// TwinCAT 3 PLC project Solutions
// ProgramVersion: 3.1.4026.11
// libraries:
//   CNM_AbstractObject, * (ekvip automation GmbH)
//   CNM AoC Lib, * (ekvip automation GmbH)
//   CNM_AssertionInterfaceLib, * (ekvip automation GmbH)
//   CNM_CollectionInterfaces, * (ekvip automation GmbH)
//   CNM_Collections, * (ekvip automation GmbH)
//   CNM_CycleManager, * (ekvip automation GmbH)
//   CNM_CylceManagerInterfaces, * (ekvip automation GmbH)
//   CNM_ReturnTypes, * (ekvip automation GmbH)
//   CNM_UnicodeUtilities, * (ekvip automation GmbH)
//   Tc2_Standard, * (Beckhoff Automation GmbH)
//   Tc2_System, * (Beckhoff Automation GmbH)
// project tree:
//   Day01/ Day01Solution.TcPOU
//   Day02/ Day02Solution.TcPOU
//   Day06/Guard/ Guard.TcPOU, IGuard.TcIO
//   Day06/Moves/ GuardMove.TcPOU, IMove.TcIO, MoveUp.TcPOU, MoveRight.TcPOU, MoveDown.TcPOU, MoveLeft.TcPOU
//   Day06/ Rotation.TcDUT, Day06Solution.TcPOU
//   Day07/ Day07Solution.TcPOU
//   Day05/ Day05Solution.TcPOU, IPage.TcIO, Page.TcPOU
//   Day04/ CharObj.TcPOU, Day04Solution.TcPOU, IChar.TcIO
//   Day03/ Day03Solution.TcPOU, DontInstruction.TcPOU, ISumCollectorLINT.TcIO, MulInstruction.TcPOU, DoInstruction.TcPOU, SumCollectorLINT.TcPOU
//   Helpers/DynArray/ Dynamic2dArray.TcPOU, I2dArray.TcIO
//   Parsers/ NumberParser.TcPOU
//   / PlcTask.TcTTO
//   POUs/ LocalIoAddresses.TcGVL, MAIN.TcPOU
// real-time tasks:
//   TASK PlcTask: cycle T#10ms, priority 20, ADS port 350

CONFIGURATION Solutions
    RESOURCE PLC ON TwinCAT3
        TASK PlcTask(INTERVAL := T#10ms, PRIORITY := 20);
        PROGRAM MAIN WITH PlcTask : MAIN;
    END_RESOURCE
END_CONFIGURATION

// ---- Day06/Rotation.TcDUT
{attribute 'qualified_only'}
{attribute 'strict'}
TYPE Rotation :
(
	UP := 0,
	RIGHT := 1,
	DOWN := 2,
	LEFT := 3
)DINT;
END_TYPE

// ---- POUs/LocalIoAddresses.TcGVL
{attribute 'qualified_only'}
VAR_GLOBAL
	NetId :STRING := '10.175.16.49.1.1';
	Path :STRING := 'C:\Users\tdie\Documents\tdie_AOC\2024';
END_VAR

// ---- Day06/Guard/IGuard.TcIO
INTERFACE IGuard

PROPERTY direction : Rotation
GET
END_GET
SET
END_SET
END_PROPERTY

METHOD walk
VAR_INPUT
	map :I2dArray;
END_VAR
END_METHOD

PROPERTY x : DINT
GET
END_GET
SET
END_SET
END_PROPERTY

PROPERTY y : DINT
GET
END_GET
SET
END_SET
END_PROPERTY

END_INTERFACE

// ---- Day06/Moves/IMove.TcIO
INTERFACE IMove

METHOD tryMove : BOOL
VAR_INPUT
	guard :IGuard;
	map :I2dArray;
	collision :DINT := 1;
END_VAR
END_METHOD

END_INTERFACE

// ---- Day03/ISumCollectorLINT.TcIO
INTERFACE ISumCollectorLINT EXTENDS CNM_AbstractObject.IObject

METHOD addValue
VAR_INPUT
	value :LINT;
END_VAR
END_METHOD

PROPERTY enabled : BOOL
GET
END_GET
SET
END_SET
END_PROPERTY

PROPERTY sum : LINT
GET
END_GET
SET
END_SET
END_PROPERTY

END_INTERFACE

// ---- Day04/IChar.TcIO
INTERFACE IChar EXTENDS IObject

PROPERTY charAsByte : Byte
GET
END_GET
END_PROPERTY

PROPERTY charAsString : STRING(1)
GET
END_GET
END_PROPERTY

END_INTERFACE

// ---- Day05/IPage.TcIO
INTERFACE IPage EXTENDS IObject, CNM_AoC.IHaveValue

METHOD addSuccessor
VAR_INPUT
	successor :CNM_AoC.IHaveValue;
END_VAR
END_METHOD

END_INTERFACE

// ---- Helpers/DynArray/I2dArray.TcIO
INTERFACE I2dArray EXTENDS CNM_AbstractObject.IObject

METHOD getObjectAt : IObject
VAR_INPUT
	y :UDINT; //dimension 1
	x :UDINT; //dimension 2
END_VAR
END_METHOD

METHOD isInBounds : BOOL
VAR_INPUT
	x :UDINT;
	y :UDINT;
END_VAR
END_METHOD

METHOD setObjectAt
VAR_INPUT
	y :UDINT; //dimension 1
	x :UDINT; //dimension 2
	obj :CNM_AbstractObject.IObject;
END_VAR
END_METHOD

END_INTERFACE

// ---- POUs/MAIN.TcPOU
PROGRAM MAIN
VAR
	day01 :Day01Solution(sNetId := LocalIoAddresses.NetId, folderPath := LocalIoAddresses.Path, inputFile := 'day01.txt', outputFile := 'solution.txt');
	day02 :Day02Solution(sNetId := LocalIoAddresses.NetId, folderPath := LocalIoAddresses.Path, inputFile := 'day02.txt', outputFile := 'solution.txt');
	day03 :Day03Solution(sNetId := LocalIoAddresses.NetId, folderPath := LocalIoAddresses.Path, inputFile := 'day03.txt', outputFile := 'solution.txt');
	day04 :Day04Solution(sNetId := LocalIoAddresses.NetId, folderPath := LocalIoAddresses.Path, inputFile := 'day04.txt', outputFile := 'solution.txt');
	day05 :Day05Solution(sNetId := LocalIoAddresses.NetId, folderPath := LocalIoAddresses.Path, inputFile := 'day05.txt', outputFile := 'solution.txt');
	day06 :Day06Solution(sNetId := LocalIoAddresses.NetId, folderPath := LocalIoAddresses.Path, inputFile := 'day06.txt', outputFile := 'solution.txt');
	day07 :Day07Solution(sNetId := LocalIoAddresses.NetId, folderPath := LocalIoAddresses.Path, inputFile := 'day07.txt', outputFile := 'solution.txt');
END_VAR

//some are really slow because I do to few operations each cycle, might take up to 30 seconds to complete!
day01.run(FALSE);
day02.run(FALSE);
day03.run(FALSE); 
day04.run(FALSE); 
day05.run(FALSE); 
day06.run(FALSE); 
day07.run(FALSE);

END_PROGRAM

// ---- Day01/Day01Solution.TcPOU
FUNCTION_BLOCK Day01Solution EXTENDS CNM_AoC.AbstractSolver

METHOD solve
VAR_INPUT
	step	: DINT;
END_VAR
VAR_INST
	pathInserted :BOOL;
	left :CNM_Collections.ArrayList(100);
	right :CNM_Collections.ArrayList(100);
	parser :NumberParser();
	sum : DINT;
END_VAR
VAR
	parsed :CNM_CollectionInterfaces.IArrayList;
	tmpObj :CNM_AbstractObject.IObject;
	value1 :CNM_AoC.IHaveValue;
	value2 :CNM_AoC.IHaveValue;
	index : DINT;
	currentLine :ILine;
	currentLineObject :IObject;
END_VAR
VAR CONSTANT
	READ_INPUT :DINT := 2;
	GET_LINES :DINT := READ_INPUT + 1;
	PARSE :DINT := GET_LINES + 1;
	SORT_LEFT :DINT := PARSE + 1;
	SORT_RIGHT :DINT := SORT_LEFT + 1;
	SOLVE_PART1 :DINT := SORT_RIGHT + 1;
	RESET_FOR_PART2 :DINT := SOLVE_PART1 + 1;
	SOLVE_PART2 :DINT := RESET_FOR_PART2 + 1;
	APPEND_SOLUTION :DINT := SOLVE_PART2 + 1;
	WRITE_SOLUTION :DINT := APPEND_SOLUTION + 1;
	CLEAN_UP :DINT := WRITE_SOLUTION + 1;
END_VAR
CASE step OF
PARSE:	
	THIS^.lines.iterate(execute := FALSE);
	WHILE(THIS^.lines.iterate(execute := TRUE, line => currentLine) = CNM_ReturnTypes.SingleExecutionState.BUSY)DO
		parsed := parser.getAllNumbers(currentLine);
		left.append(parsed.dequeue());
		right.append(parsed.dequeue());
		parsed.deepDestruct();
	END_WHILE
	cm.proceed();
SORT_LEFT:
	cm.evaluate(SEL(right.size = left.size, CNM_ReturnTypes.SingleExecutionState.ERROR, CNM_ReturnTypes.SingleExecutionState.SUCCESS));
	cm.evaluate(left.instant.sort());
SORT_RIGHT:
	cm.evaluate(right.instant.sort());
SOLVE_PART1:
	FOR index := 0 TO TO_DINT(left.size)-1 DO
		left.getObjectAt(index, object => tmpObj);
		__QUERYINTERFACE(tmpObj, value1);
		right.getObjectAt(index, object => tmpObj);
		__QUERYINTERFACE(tmpObj, value2);
		sum := sum + TO_DINT(ABS(value1.value - value2.value));
	END_FOR
	THIS^.bufferWrite := Concat(TO_STRING(sum), '$n');
	cm.proceed();
RESET_FOR_PART2:
	left.iterate(FALSE);
	sum := 0;
	cm.proceed();
SOLVE_PART2:
	cm.evaluate(left.iterate(TRUE, object => tmpObj));
	IF(__QUERYINTERFACE(tmpObj, value1))THEN
		right.iterate(FALSE);
		WHILE(right.iterate(TRUE, object => tmpObj) = CNM_ReturnTypes.SingleExecutionState.BUSY AND __QUERYINTERFACE(tmpObj, value2))DO
			IF(value1.value = value2.value)THEN
				sum := sum + TO_DINT(value1.value);
			END_IF
			IF(value2.value > value1.value)THEN
				EXIT;
			END_IF
		END_WHILE
	END_IF		
APPEND_SOLUTION:
	THIS^.bufferWrite :=Concat(THIS^.bufferWrite, Concat(TO_STRING(sum), '$n'));
	cm.proceed();
WRITE_SOLUTION:
	THIS^.writeSolution();
CLEAN_UP:
	cm.step.next := CNM_ReturnTypes.DefaultSteps.STEP.SUCCESS;
	lines.deepDestruct();
	left.deepDestruct();
	right.deepDestruct();
	cm.proceed();
END_CASE
END_METHOD

END_FUNCTION_BLOCK

// ---- Parsers/NumberParser.TcPOU
FUNCTION_BLOCK NumberParser
VAR_INPUT
END_VAR
VAR_OUTPUT
END_VAR
VAR
END_VAR

METHOD getAllNumbers : IArrayList
VAR_INPUT
	container :CNM_AoC.IStringContainer;
END_VAR
VAR
	index : DINT;
	currentParseValue :DINT;
	currentLineText : STRING(255);
	found :BOOL;
	result :CNM_CollectionInterfaces.IArrayList;
	pResult :POINTER TO CNM_Collections.ArrayList;
	pValue :POINTER TO CNM_AoC.Value;
	value :CNM_AoC.IHaveValue;
END_VAR
pResult := __NEW(ArrayList(initialSize := 2));
__QUERYINTERFACE(pResult^, result);
currentLineText := container.text;

FOR index := 0 TO LEN(container.text)-1 DO
	IF(currentLineText[index] >= 48 AND currentLineText[index] <= 57)THEN
		currentParseValue := currentParseValue * 10;
		currentParseValue := currentParseValue + currentLineText[index]-48;
		found := TRUE;
	ELSE
		IF(found)THEN
			pValue := __NEW(Value);
			__QUERYINTERFACE(pValue^, value);
			value.value := currentParseValue;//add num to result
			result.append(value);
		END_IF
		currentParseValue := 0;
		found := FALSE;
	END_IF
END_FOR	

IF(found)THEN
	pValue := __NEW(Value);
	__QUERYINTERFACE(pValue^, value);
	value.value := currentParseValue;//add num to result
	result.append(value);
END_IF

getAllNumbers := result;
END_METHOD

METHOD getAllNumbersLint : IArrayList
VAR_INPUT
	container :CNM_AoC.IStringContainer;
END_VAR
VAR
	index : DINT;
	currentParseValue :LINT;
	currentLineText : STRING(255);
	found :BOOL;
	result :CNM_CollectionInterfaces.IArrayList;
	pResult :POINTER TO CNM_Collections.ArrayList;
	pValue :POINTER TO CNM_AoC.LintValue;
	value :CNM_AoC.IHaveLintValue;
END_VAR
pResult := __NEW(ArrayList(initialSize := 2));
__QUERYINTERFACE(pResult^, result);
currentLineText := container.text;

FOR index := 0 TO LEN(container.text)-1 DO
	IF(currentLineText[index] >= 48 AND currentLineText[index] <= 57)THEN
		currentParseValue := currentParseValue * 10;
		currentParseValue := currentParseValue + currentLineText[index]-48;
		found := TRUE;
	ELSE
		IF(found)THEN
			pValue := __NEW(LintValue);
			__QUERYINTERFACE(pValue^, value);
			value.value := currentParseValue;//add num to result
			result.append(value);
		END_IF
		currentParseValue := 0;
		found := FALSE;
	END_IF
END_FOR	

IF(found)THEN
	pValue := __NEW(LintValue);
	__QUERYINTERFACE(pValue^, value);
	value.value := currentParseValue;//add num to result
	result.append(value);
END_IF

getAllNumbersLint := result;
END_METHOD

METHOD getAllNumbersUlint : IArrayList
VAR_INPUT
	container :CNM_AoC.IStringContainer;
END_VAR
VAR
	index : DINT;
	currentParseValue :ULINT;
	currentLineText : STRING(255);
	found :BOOL;
	result :CNM_CollectionInterfaces.IArrayList;
	pResult :POINTER TO CNM_Collections.ArrayList;
	pValue :POINTER TO CNM_AoC.UlintValue;
	value :CNM_AoC.IHaveUlintValue;
END_VAR
pResult := __NEW(ArrayList(initialSize := 2));
__QUERYINTERFACE(pResult^, result);
currentLineText := container.text;

FOR index := 0 TO LEN(container.text)-1 DO
	IF(currentLineText[index] >= 48 AND currentLineText[index] <= 57)THEN
		currentParseValue := currentParseValue * 10;
		currentParseValue := currentParseValue + currentLineText[index]-48;
		found := TRUE;
	ELSE
		IF(found)THEN
			pValue := __NEW(UlintValue);
			__QUERYINTERFACE(pValue^, value);
			value.value := currentParseValue;//add num to result
			result.append(value);
		END_IF
		currentParseValue := 0;
		found := FALSE;
	END_IF
END_FOR	

IF(found)THEN
	pValue := __NEW(UlintValue);
	__QUERYINTERFACE(pValue^, value);
	value.value := currentParseValue;//add num to result
	result.append(value);
END_IF

getAllNumbersUlint := result;
END_METHOD

END_FUNCTION_BLOCK

// ---- Day02/Day02Solution.TcPOU
FUNCTION_BLOCK Day02Solution EXTENDS AbstractSolver

METHOD PRIVATE isSequenceValid : BOOL
VAR_INPUT
	sequence :CNM_CollectionInterfaces.IArrayList;
END_VAR
VAR
	tmpObj :CNM_AbstractObject.IObject;
	number :CNM_AoC.IHaveValue;
	skipped : BOOL;
	first :BOOL;
	second :BOOL;
	lastValue :DINT;
	prevLastValue :DINT := -1;
	errors :DINT := 0;
	currentValue :DINT;
	sequenceResult :CNM_ReturnTypes.SingleExecutionState;
	order :DINT; //-1 falling, 1 rising, 0 unknown
END_VAR
sequence.iterate(FALSE);
WHILE((sequenceResult := sequence.iterate(TRUE, object => tmpObj)) = CNM_ReturnTypes.SingleExecutionState.BUSY AND __QUERYINTERFACE(tmpObj, number))DO
	currentValue := TO_DINT(number.value);
	IF(NOT first)THEN
		lastValue := currentValue;
		first := TRUE;
		CONTINUE;
	END_IF
	IF(ABS(currentValue - lastValue) > 3 OR ABS(currentValue - lastValue) = 0)THEN
		EXIT;
	END_IF
	IF(currentValue > lastValue)THEN
		IF(order = -1)THEN
			EXIT;
		ELSE
			order := 1;
		END_IF
	END_IF
	IF(currentValue < lastValue)THEN
		IF(order = 1)THEN
			EXIT;
		ELSE
			order := -1;
		END_IF
	END_IF
	lastValue := currentValue;
END_WHILE
isSequenceValid := (sequenceResult = CNM_ReturnTypes.SingleExecutionState.SUCCESS);
END_METHOD

METHOD solve
VAR_INPUT
	step	: DINT;
END_VAR
VAR_INST
	pathInserted :BOOL;
	sequences :CNM_Collections.ArrayList(100);
	parser :NumberParser();
	sum : DINT;
END_VAR
VAR
	parsed :CNM_CollectionInterfaces.IArrayList;
	tmpObj :CNM_AbstractObject.IObject;
	sequence :CNM_CollectionInterfaces.IArrayList;
	sequenceCopy :CNM_CollectionInterfaces.IArrayList;
	index : DINT;
	currentLine :ILine;
	currentLineObject :IObject;
END_VAR
VAR CONSTANT
	READ_INPUT :DINT := 2;
	GET_LINES :DINT := READ_INPUT + 1;
	PARSE :DINT := GET_LINES + 1;
	SOLVE_PART1 :DINT := PARSE + 1;
	RESET_FOR_PART2 :DINT := SOLVE_PART1 + 1;
	SOLVE_PART2 :DINT := RESET_FOR_PART2 + 1;
	APPEND_SOLUTION :DINT := SOLVE_PART2 + 1;
	WRITE_SOLUTION :DINT := APPEND_SOLUTION + 1;
	CLEAN_UP :DINT := WRITE_SOLUTION + 1;
END_VAR
CASE step OF
PARSE:	
	THIS^.lines.iterate(execute := FALSE);
	WHILE(THIS^.lines.iterate(execute := TRUE, line => currentLine) = CNM_ReturnTypes.SingleExecutionState.BUSY)DO
		parsed := parser.getAllNumbers(currentLine);
		sequences.append(parsed);
	END_WHILE
	cm.proceed();	
SOLVE_PART1:
	cm.evaluate(sequences.iterate(cm.executeStep, object => tmpObj));
	IF(__QUERYINTERFACE(tmpObj, sequence))THEN
		IF(THIS^.isSequenceValid(sequence))THEN
			sum := sum + 1;
		END_IF
	END_IF		
RESET_FOR_PART2:
	THIS^.bufferWrite := Concat(TO_STRING(sum), '$n');
	sum := 0;
	cm.proceed();
SOLVE_PART2:
	cm.evaluate(sequences.iterate(cm.executeStep, object => tmpObj));
	IF(__QUERYINTERFACE(tmpObj, sequence))THEN
		FOR index := 0 TO TO_DINT(sequence.size)-1 DO
			IF(sequence.clone(clonedObject => tmpObj) = CNM_ReturnTypes.CloneResult.SUCCESS AND_THEN __QUERYINTERFACE(tmpObj, sequenceCopy))THEN
				sequenceCopy.removeObjectAt(index);
				IF(THIS^.isSequenceValid(sequenceCopy))THEN
					sum := sum + 1;
					sequenceCopy.destruct();
					EXIT;
				END_IF
				sequenceCopy.destruct();
			END_IF
		END_FOR
	END_IF		
APPEND_SOLUTION:
	THIS^.bufferWrite :=Concat(THIS^.bufferWrite, Concat(TO_STRING(sum), '$n'));
	cm.proceed();
WRITE_SOLUTION:
	THIS^.writeSolution();
CLEAN_UP:
	cm.step.next := CNM_ReturnTypes.DefaultSteps.STEP.SUCCESS;
	lines.deepDestruct();
	sequences.deepDestruct();
	cm.proceed();
END_CASE
END_METHOD

END_FUNCTION_BLOCK

// ---- Day03/Day03Solution.TcPOU
FUNCTION_BLOCK Day03Solution EXTENDS AbstractSolver
VAR
	sumCollector :SumCollectorLINT();
END_VAR

METHOD solve
VAR_INPUT
	step	: DINT;
END_VAR
VAR_INST
	pathInserted :BOOL;
	instructions :CNM_Collections.ArrayList(100);
END_VAR
VAR
	parsed :CNM_CycleManagerInterfaces.ISingleAttempt;	
	tmpObj :CNM_AbstractObject.IObject;
	instruction :CNM_CycleManagerInterfaces.ISingleAttempt;	
	index : UDINT;
	currentLine :ILine;
	currentLineObject :IObject;
END_VAR
VAR CONSTANT
	READ_INPUT :DINT := 2;
	GET_LINES :DINT := READ_INPUT + 1;
	PARSE :DINT := GET_LINES + 1;
	SOLVE_PART1 :DINT := PARSE + 1;
	RESET_FOR_PART2 :DINT := SOLVE_PART1 + 1;
	SOLVE_PART2 :DINT := RESET_FOR_PART2 + 1;
	APPEND_SOLUTION :DINT := SOLVE_PART2 + 1;
	WRITE_SOLUTION :DINT := APPEND_SOLUTION + 1;
	CLEAN_UP :DINT := WRITE_SOLUTION + 1;
END_VAR
CASE step OF
PARSE:	
	FOR(index := 0) TO SIZEOF(THIS^.bufferRead) DO
		IF(THIS^.bufferRead[index] = 0)THEN
			EXIT;
		END_IF
		IF(THIS^.tryParseInstruction(ADR(THIS^.bufferRead), SIZEOF(THIS^.bufferRead), index, instruction => parsed))THEN			
			instructions.append(parsed);
		END_IF			
	END_FOR
	cm.proceed();	
SOLVE_PART1:
	cm.evaluate(instructions.iterate(cm.executeStep, object => tmpObj));
	IF(__QUERYINTERFACE(tmpObj, instruction))THEN
		IF(instruction.className = 'MulInstruction')THEN
			instruction.invoke();
		END_IF
	END_IF		
RESET_FOR_PART2:
	THIS^.bufferWrite := Concat(TO_STRING(sumCollector.sum), '$n');
	sumCollector.sum := 0;
	cm.proceed();
SOLVE_PART2:
	cm.evaluate(instructions.iterate(cm.executeStep, object => tmpObj));
	IF(__QUERYINTERFACE(tmpObj, instruction))THEN
		instruction.invoke();
	END_IF		
APPEND_SOLUTION:
	THIS^.bufferWrite :=Concat(THIS^.bufferWrite, Concat(TO_STRING(sumCollector.sum), '$n'));
	cm.proceed();
WRITE_SOLUTION:
	THIS^.writeSolution();
CLEAN_UP:
	cm.step.next := CNM_ReturnTypes.DefaultSteps.STEP.SUCCESS;
	lines.deepDestruct();
	instructions.deepDestruct();
	cm.proceed();
END_CASE
END_METHOD

METHOD tryParseInstruction : BOOL
VAR_INPUT
	text :POINTER TO BYTE;
	maxIndex :UDINT;
END_VAR
VAR_IN_OUT
	index :UDINT;
END_VAR
VAR_OUTPUT
	instruction :CNM_CycleManagerInterfaces.ISingleAttempt;
END_VAR
VAR CONSTANT
	mulStart :STRING :='mul(';
	doStart :STRING :='do()';
	doNotStart :STRING :='don$'t()';	
	digits :STRING :='0123456789';
	comma :STRING :=',';
	closedbracket :STRING :=')';
END_VAR
VAR
	validNum :BOOL := FALSE;
	numIndex :UDINT := 0;
	num1 :LINT;
	num2 :LINT;
	mulInst :POINTER TO MulInstruction;
	doInst :POINTER TO DoInstruction;
	doNotInst :POINTER TO DontInstruction;
END_VAR
//parsing in TwinCAT is no fun without better libraries
tryParseInstruction := FALSE;

IF(index + 8 < maxIndex 
	AND_THEN text[index] = mulStart[0] 
	AND_THEN text[index+1] = mulStart[1]
	AND_THEN text[index+2] = mulStart[2]
	AND_THEN text[index+3] = mulStart[3]
)THEN
	WHILE(index + 4 + numIndex < maxIndex AND_THEN text[index+4+numIndex] >= digits[0] AND_THEN text[index+4+numIndex] <= digits[9])DO
		validNum := TRUE;
		num1 := num1 * 10 + (text[index+4+numIndex] -48);
		numIndex := numIndex + 1;
	END_WHILE
	RETURN (NOT validNum);
	RETURN (text[index+4+numIndex] <> comma[0]);
	numIndex := numIndex + 1;
	validNum := FALSE;
	WHILE(index + 4 + numIndex < maxIndex AND_THEN text[index+4+numIndex] >= digits[0] AND_THEN text[index+4+numIndex] <= digits[9])DO
		validNum := TRUE;
		num2 := num2 * 10 + (text[index+4+numIndex] -48);
		numIndex := numIndex + 1;
	END_WHILE
	RETURN (NOT validNum);
	RETURN (text[index+4+numIndex] <> closedbracket[0]);
	mulInst := __NEW(MulInstruction(left := num1, right := num2, collector := THIS^.sumCollector));
	RETURN (NOT __QUERYINTERFACE(mulInst^, instruction));
	tryParseInstruction := TRUE;
ELSIF(index + 7 < maxIndex 
	AND_THEN text[index] = doNotStart[0] 
	AND_THEN text[index+1] = doNotStart[1]
	AND_THEN text[index+2] = doNotStart[2]
	AND_THEN text[index+3] = doNotStart[3]
	AND_THEN text[index+4] = doNotStart[4]
	AND_THEN text[index+5] = doNotStart[5]
	AND_THEN text[index+6] = doNotStart[6]
)THEN
	doNotInst := __NEW(DontInstruction(collector := THIS^.sumCollector));
	RETURN (NOT __QUERYINTERFACE(doNotInst^, instruction));
	tryParseInstruction := TRUE;
ELSIF(index + 7 < maxIndex 
	AND_THEN text[index] = doStart[0] 
	AND_THEN text[index+1] = doStart[1]
	AND_THEN text[index+2] = doStart[2]
	AND_THEN text[index+3] = doStart[3]
)THEN
	doInst := __NEW(DoInstruction(collector := THIS^.sumCollector));
	RETURN (NOT __QUERYINTERFACE(doInst^, instruction));
	tryParseInstruction := TRUE;
END_IF
END_METHOD

END_FUNCTION_BLOCK

// ---- Day03/SumCollectorLINT.TcPOU
{attribute 'enable_dynamic_creation'}
FUNCTION_BLOCK SumCollectorLINT EXTENDS Object IMPLEMENTS ISumCollectorLINT
VAR
	isEnabled :BOOL := TRUE;
	myValue :LINT := 0;
END_VAR

METHOD addValue
VAR_INPUT
	value	: LINT;
END_VAR
RETURN (NOT THIS^.enabled);
THIS^.myValue := THIS^.myValue + value;
END_METHOD

(*

short summary
=================
This abstract property returns the class name of the concrete object, 
which is useful for logging/debugging purpose or to check the class name
for ``__DELETE`` in factories (sometimes it's necessary to do more 
than just to free the memory).

.. <legal notes>

legal notes
=================
| SPDX-FileCopyrightText: © 2022 ekvip automation GmbH <info@ekvip.de>
| SPDX-License-Identifier: Apache-2.0
| For details check: Apache-2.0_

.. _Apache-2.0: https://www.apache.org/licenses/LICENSE-2.0

.. </legal notes>

*)
PROPERTY className : CNM_AbstractObject.ClassName
GET
className := 'SumCollectorLINT';
END_GET
END_PROPERTY

PROPERTY enabled : BOOL
GET
enabled := THIS^.isEnabled;
END_GET
SET
THIS^.isEnabled := enabled;
END_SET
END_PROPERTY

{warning 'Add property implementation'}
PROPERTY sum : LINT
GET
sum := THIS^.myValue;
END_GET
SET
THIS^.myValue := sum;
END_SET
END_PROPERTY

END_FUNCTION_BLOCK

// ---- Day03/MulInstruction.TcPOU
{attribute 'enable_dynamic_creation'}
FUNCTION_BLOCK MulInstruction EXTENDS Object IMPLEMENTS ISingleAttempt
VAR
	myLeft :LINT;
	myRight :LINT;
	myCollector :ISumCollectorLINT;
END_VAR

{warning 'Add property implementation'}
(*

short summary
=================
This abstract property returns the class name of the concrete object, 
which is useful for logging/debugging purpose or to check the class name
for ``__DELETE`` in factories (sometimes it's necessary to do more 
than just to free the memory).

.. <legal notes>

legal notes
=================
| SPDX-FileCopyrightText: © 2022 ekvip automation GmbH <info@ekvip.de>
| SPDX-License-Identifier: Apache-2.0
| For details check: Apache-2.0_

.. _Apache-2.0: https://www.apache.org/licenses/LICENSE-2.0

.. </legal notes>

*)
PROPERTY className : CNM_AbstractObject.ClassName
GET
className := 'MulInstruction';
END_GET
END_PROPERTY

//FB_Init is always available implicitly and it is used primarily for initialization.
//The return value is not evaluated. For a specific influence, you can also declare the
//methods explicitly and provide additional code there with the standard initialization
//code. You can evaluate the return value.
METHOD FB_Init: BOOL
VAR_INPUT
    bInitRetains: BOOL; // TRUE: the retain variables are initialized (reset warm / reset cold)
    bInCopyCode: BOOL;  // TRUE: the instance will be copied to the copy code afterward (online change)   
	left :LINT;
	right :LINT;
	collector :ISumCollectorLINT;
END_VAR
THIS^.myLeft := left;
THIS^.myRight := right;
THIS^.myCollector := collector;
END_METHOD

(*

short summary
=================
Invokes the action associated with this interface.

.. <legal notes>

legal notes
=================
| SPDX-FileCopyrightText: © 2024 ekvip automation GmbH <info@ekvip.de>
| SPDX-License-Identifier: Apache-2.0
| For details check: Apache-2.0_

.. _Apache-2.0: https://www.apache.org/licenses/LICENSE-2.0

.. </legal notes>

parameters
=================

*)
METHOD invoke : CNM_CycleManagerInterfaces.CNM_ReturnTypes.SingleExecutionResult
THIS^.myCollector.addValue(THIS^.myLeft * THIS^.myRight);
END_METHOD

END_FUNCTION_BLOCK

// ---- Day03/DoInstruction.TcPOU
{attribute 'enable_dynamic_creation'}
FUNCTION_BLOCK DoInstruction EXTENDS Object IMPLEMENTS ISingleAttempt
VAR
	myCollector :ISumCollectorLINT;
END_VAR

{warning 'Add property implementation'}
(*

short summary
=================
This abstract property returns the class name of the concrete object, 
which is useful for logging/debugging purpose or to check the class name
for ``__DELETE`` in factories (sometimes it's necessary to do more 
than just to free the memory).

.. <legal notes>

legal notes
=================
| SPDX-FileCopyrightText: © 2022 ekvip automation GmbH <info@ekvip.de>
| SPDX-License-Identifier: Apache-2.0
| For details check: Apache-2.0_

.. _Apache-2.0: https://www.apache.org/licenses/LICENSE-2.0

.. </legal notes>

*)
PROPERTY className : CNM_AbstractObject.ClassName
GET
className := 'DoInstruction';
END_GET
END_PROPERTY

//FB_Init is always available implicitly and it is used primarily for initialization.
//The return value is not evaluated. For a specific influence, you can also declare the
//methods explicitly and provide additional code there with the standard initialization
//code. You can evaluate the return value.
METHOD FB_Init: BOOL
VAR_INPUT
    bInitRetains: BOOL; // TRUE: the retain variables are initialized (reset warm / reset cold)
    bInCopyCode: BOOL;  // TRUE: the instance will be copied to the copy code afterward (online change)   
	collector :ISumCollectorLINT;
END_VAR
THIS^.myCollector := collector;
END_METHOD

(*

short summary
=================
Invokes the action associated with this interface.

.. <legal notes>

legal notes
=================
| SPDX-FileCopyrightText: © 2024 ekvip automation GmbH <info@ekvip.de>
| SPDX-License-Identifier: Apache-2.0
| For details check: Apache-2.0_

.. _Apache-2.0: https://www.apache.org/licenses/LICENSE-2.0

.. </legal notes>

parameters
=================

*)
METHOD invoke : CNM_CycleManagerInterfaces.CNM_ReturnTypes.SingleExecutionResult
THIS^.myCollector.enabled := TRUE;
END_METHOD

END_FUNCTION_BLOCK

// ---- Day03/DontInstruction.TcPOU
{attribute 'enable_dynamic_creation'}
FUNCTION_BLOCK DontInstruction EXTENDS Object IMPLEMENTS ISingleAttempt
VAR
	myCollector :ISumCollectorLINT;
END_VAR

{warning 'Add property implementation'}
(*

short summary
=================
This abstract property returns the class name of the concrete object, 
which is useful for logging/debugging purpose or to check the class name
for ``__DELETE`` in factories (sometimes it's necessary to do more 
than just to free the memory).

.. <legal notes>

legal notes
=================
| SPDX-FileCopyrightText: © 2022 ekvip automation GmbH <info@ekvip.de>
| SPDX-License-Identifier: Apache-2.0
| For details check: Apache-2.0_

.. _Apache-2.0: https://www.apache.org/licenses/LICENSE-2.0

.. </legal notes>

*)
PROPERTY className : CNM_AbstractObject.ClassName
GET
className := 'DontInstruction';
END_GET
END_PROPERTY

//FB_Init is always available implicitly and it is used primarily for initialization.
//The return value is not evaluated. For a specific influence, you can also declare the
//methods explicitly and provide additional code there with the standard initialization
//code. You can evaluate the return value.
METHOD FB_Init: BOOL
VAR_INPUT
    bInitRetains: BOOL; // TRUE: the retain variables are initialized (reset warm / reset cold)
    bInCopyCode: BOOL;  // TRUE: the instance will be copied to the copy code afterward (online change)   
	collector :ISumCollectorLINT;
END_VAR
THIS^.myCollector := collector;
END_METHOD

(*

short summary
=================
Invokes the action associated with this interface.

.. <legal notes>

legal notes
=================
| SPDX-FileCopyrightText: © 2024 ekvip automation GmbH <info@ekvip.de>
| SPDX-License-Identifier: Apache-2.0
| For details check: Apache-2.0_

.. _Apache-2.0: https://www.apache.org/licenses/LICENSE-2.0

.. </legal notes>

parameters
=================

*)
METHOD invoke : CNM_CycleManagerInterfaces.CNM_ReturnTypes.SingleExecutionResult
THIS^.myCollector.enabled := FALSE;
END_METHOD

END_FUNCTION_BLOCK

// ---- Day04/Day04Solution.TcPOU
FUNCTION_BLOCK Day04Solution EXTENDS AbstractSolver
VAR	
	xmases :I2dArray;
	sizeY :UDINT;
	sizeX :UDINT;
END_VAR

METHOD countXMAS : DINT
VAR_INPUT
	x :UDINT;
	y :UDINT;
END_VAR
VAR
	char :IChar;
	index :UDINT;
	valids :ARRAY[0..7] OF BOOL := [8(TRUE)];
END_VAR
VAR CONSTANT
	xmas :STRING(4) := 'XMAS';
END_VAR
countXMAS := 0;

RETURN (NOT THIS^.isInBounds(x,y));
RETURN (NOT __QUERYINTERFACE(THIS^.xmases.getObjectAt(y := y, x := x), char));
RETURN ((char.charAsByte <> xmas[0]));

FOR index := 1 TO 3 DO
	valids[0] := valids[0] AND_THEN THIS^.isInBounds(x + index, y) 			AND_THEN toChar(THIS^.xmases.getObjectAt(y,x + index)).charAsByte = xmas[index];
	valids[1] := valids[1] AND_THEN THIS^.isInBounds(x + index, y + index) 	AND_THEN toChar(THIS^.xmases.getObjectAt(y + index,x + index)).charAsByte = xmas[index];
	valids[7] := valids[7] AND_THEN THIS^.isInBounds(y + index,x) 			AND_THEN toChar(THIS^.xmases.getObjectAt(y + index,x)).charAsByte = xmas[index];
	valids[4] := valids[4] AND_THEN THIS^.isInBounds(x - index, y + index)	AND_THEN toChar(THIS^.xmases.getObjectAt(y + index,x - index)).charAsByte = xmas[index];
	valids[2] := valids[2] AND_THEN THIS^.isInBounds(x - index, y) 			AND_THEN toChar(THIS^.xmases.getObjectAt(y,x - index)).charAsByte = xmas[index];
	valids[3] := valids[3] AND_THEN THIS^.isInBounds(x - index, y - index) 	AND_THEN toChar(THIS^.xmases.getObjectAt(y - index,x - index)).charAsByte = xmas[index];
	valids[6] := valids[6] AND_THEN THIS^.isInBounds(x, y - index) 			AND_THEN toChar(THIS^.xmases.getObjectAt(y - index,x)).charAsByte = xmas[index];
	valids[5] := valids[5] AND_THEN THIS^.isInBounds(x + index, y - index) 	AND_THEN toChar(THIS^.xmases.getObjectAt(y - index,x + index)).charAsByte = xmas[index];
END_FOR

FOR index := 0 TO 7 DO
	IF(valids[index])THEN
		countXMAS := countXMAS + 1;
	END_IF
END_FOR
END_METHOD

METHOD isInBounds : BOOL
VAR_INPUT
	x :UDINT;
	y :UDINT;
END_VAR
isInBounds := (x < THIS^.sizeX AND y < THIS^.sizeY); //cheat >= 0 by UDINT overflow
END_METHOD

METHOD isX : BOOL
VAR_INPUT
	x :UDINT;
	y :UDINT;
END_VAR
VAR
	char :IChar;
	index :UDINT;
END_VAR
VAR CONSTANT
	xmas :STRING(4) := 'XMAS';
END_VAR
RETURN (NOT THIS^.isInBounds(x,y));
RETURN (NOT __QUERYINTERFACE(THIS^.xmases.getObjectAt(y := y, x := x), char));
RETURN ((char.charAsByte <> xmas[2]));
RETURN (NOT (THIS^.isInBounds(x-1,y-1) AND THIS^.isInBounds(x+1,y-1) AND THIS^.isInBounds(x-1,y+1) AND THIS^.isInBounds(x+1,y+1)));

isX := (
			(toChar(THIS^.xmases.getObjectAt(y + 1,x + 1)).charAsString = 'M' 
			AND_THEN toChar(THIS^.xmases.getObjectAt(y -1 ,x - 1)).charAsString = 'S')
		OR
			(toChar(THIS^.xmases.getObjectAt(y + 1,x + 1)).charAsString = 'S' 
			AND_THEN toChar(THIS^.xmases.getObjectAt(y -1 ,x - 1)).charAsString = 'M')
	) AND (
			(toChar(THIS^.xmases.getObjectAt(y + 1,x - 1)).charAsString = 'M' 
			AND_THEN toChar(THIS^.xmases.getObjectAt(y -1 ,x + 1)).charAsString = 'S')
		OR
			(toChar(THIS^.xmases.getObjectAt(y + 1,x - 1)).charAsString = 'S' 
			AND_THEN toChar(THIS^.xmases.getObjectAt(y -1 ,x + 1)).charAsString = 'M')
	);
END_METHOD

METHOD solve
VAR_INPUT
	step	: DINT;
END_VAR
VAR_INST
	pathInserted :BOOL;
	sum : DINT;
END_VAR
VAR
	lineText :Tc2_System.T_MaxString;
	tmpObj :CNM_AbstractObject.IObject;
	char :IChar;
	pChar :POINTER TO CharObj;
	pXmas :POINTER TO Dynamic2dArray;
	curChar :STRING(1);
	index : DINT;
	indexY : DINT;
	currentLine :ILine;
	currentLineObject :IObject;
END_VAR
VAR CONSTANT
	READ_INPUT :DINT := 2;
	GET_LINES :DINT := READ_INPUT + 1;
	PARSE :DINT := GET_LINES + 1;
	SOLVE_PART1 :DINT := PARSE + 1;
	RESET_FOR_PART2 :DINT := SOLVE_PART1 + 1;
	SOLVE_PART2 :DINT := RESET_FOR_PART2 + 1;
	APPEND_SOLUTION :DINT := SOLVE_PART2 + 1;
	WRITE_SOLUTION :DINT := APPEND_SOLUTION + 1;
	CLEAN_UP :DINT := WRITE_SOLUTION + 1;
END_VAR
CASE step OF
PARSE:		
	lines.getLineAt(0, line => currentLine);
	sizeY := TO_UDINT(lines.size);
	sizeX := LEN(currentLine.text);
	pXmas := __NEW(Dynamic2dArray(sizeDim1 := sizeY, sizeDim2 := sizeX));
	RETURN (NOT __QUERYINTERFACE(pXmas^,xmases));
	THIS^.lines.iterate(execute := FALSE);
	indexY := 0;
	WHILE(THIS^.lines.iterate(execute := TRUE, line => currentLine) = CNM_ReturnTypes.SingleExecutionState.BUSY)DO
		FOR index := 0 TO sizeX DO
			lineText := currentLine.text;
			curChar := F_ToCHR(lineText[index]);
			pChar := __NEW(CharObj(char := curChar));
			xmases.setObjectAt(y := indexY, x := index, pChar^);
		END_FOR
		indexY := indexY+1;
	END_WHILE
	cm.proceed();	
SOLVE_PART1:
	FOR indexY := 0 TO sizeY DO
		FOR index := 0 TO sizeX DO
			sum := sum + THIS^.countXMAS(x := index, y := indexY);
		END_FOR
	END_FOR	
	cm.proceed();
RESET_FOR_PART2:
	THIS^.bufferWrite := Concat(TO_STRING(sum), '$n');
	sum := 0;
	cm.proceed();
SOLVE_PART2:
	FOR indexY := 0 TO sizeY DO
		FOR index := 0 TO sizeX DO
			sum := sum + SEL(THIS^.isX(index, indexY), 0, 1);
		END_FOR
	END_FOR		
	cm.proceed();
APPEND_SOLUTION:
	THIS^.bufferWrite :=Concat(THIS^.bufferWrite, Concat(TO_STRING(sum), '$n'));
	cm.proceed();
WRITE_SOLUTION:
	THIS^.writeSolution();
CLEAN_UP:
	cm.step.next := CNM_ReturnTypes.DefaultSteps.STEP.SUCCESS;
	lines.deepDestruct();
	xmases.deepDestruct();
	cm.proceed();
END_CASE
END_METHOD

METHOD toChar : IChar
VAR_INPUT
	obj : CNM_AbstractObject.IObject;
END_VAR
__QUERYINTERFACE(obj, toChar);
END_METHOD

END_FUNCTION_BLOCK

// ---- Day04/CharObj.TcPOU
{attribute 'enable_dynamic_creation'}
FUNCTION_BLOCK CharObj EXTENDS Object IMPLEMENTS IChar
VAR
	myChar : STRING(1);
END_VAR

PROPERTY charAsByte : Byte
GET
charAsByte := THIS^.myChar[0];
END_GET
END_PROPERTY

PROPERTY charAsString : STRING(1)
GET
charAsString := THIS^.myChar;
END_GET
END_PROPERTY

(*

short summary
=================
This abstract property returns the class name of the concrete object, 
which is useful for logging/debugging purpose or to check the class name
for ``__DELETE`` in factories (sometimes it's necessary to do more 
than just to free the memory).

.. <legal notes>

legal notes
=================
| SPDX-FileCopyrightText: © 2022 ekvip automation GmbH <info@ekvip.de>
| SPDX-License-Identifier: Apache-2.0
| For details check: Apache-2.0_

.. _Apache-2.0: https://www.apache.org/licenses/LICENSE-2.0

.. </legal notes>

*)
PROPERTY className : CNM_AbstractObject.ClassName
GET
className := 'CharObj';
END_GET
END_PROPERTY

(*

short summary
=================
The constructor ``FB_init`` is needed to create an unique hash code.
The hash code is a pseudo random number create with a xorshift_ algorithm.
It can be overwritten on derivations, because it will be called implicit, ``SUPER^.FB_init()`` is not required.
For more information check: `Behavoir with derived function blocks`_

.. _Behavoir with derived function blocks: https://infosys.beckhoff.com/content/1033/tc3_plc_intro/5482088715.html?id=6983869892358031022
.. _xorshift: https://en.wikipedia.org/wiki/Xorshift

.. <legal notes>

legal notes
=================
| SPDX-FileCopyrightText: © 2022 ekvip automation GmbH <info@ekvip.de>
| SPDX-License-Identifier: Apache-2.0
| For details check: Apache-2.0_

.. _Apache-2.0: https://www.apache.org/licenses/LICENSE-2.0

.. </legal notes>

parameters
=================

*)
METHOD FB_init : BOOL
VAR_INPUT
	(* if TRUE, the retain variables are initialized (warm start / cold start)*)
	bInitRetains	: BOOL;
	(* if TRUE, the instance afterwards gets moved into the copy code (online change) *)
	bInCopyCode	: BOOL;
	char :STRING(1);
END_VAR
THIS^.myChar := char;
END_METHOD

END_FUNCTION_BLOCK

// ---- Helpers/DynArray/Dynamic2dArray.TcPOU
{attribute 'enable_dynamic_creation'}
FUNCTION_BLOCK Dynamic2dArray EXTENDS Object IMPLEMENTS I2dArray
VAR
	dim1 :UDINT;
	dim2 :UDINT;
	container :POINTER TO CNM_AbstractObject.IObject;
END_VAR

(*

short summary
=================
This abstract property returns the class name of the concrete object, 
which is useful for logging/debugging purpose or to check the class name
for ``__DELETE`` in factories (sometimes it's necessary to do more 
than just to free the memory).

.. <legal notes>

legal notes
=================
| SPDX-FileCopyrightText: © 2022 ekvip automation GmbH <info@ekvip.de>
| SPDX-License-Identifier: Apache-2.0
| For details check: Apache-2.0_

.. _Apache-2.0: https://www.apache.org/licenses/LICENSE-2.0

.. </legal notes>

*)
PROPERTY className : CNM_AbstractObject.ClassName
GET
className := 'Dynamic2dArray';
END_GET
END_PROPERTY

(*

short summary
=================
This method is a self-destruction if the object was created dynamically.
If the object is a container class, the container content is destroyed with it.
The output NULL is a constant which is always NULL,
this allows a semi-pleasant notation: ``foo.deepDestruct(NULL => foo);``.

.. attention:: 
	For derivations: **If a derived class needs ``deepDestruct`` this method must be overwritten.**
	otherwise it just calls :ref:`Object.destruct`. 


.. <legal notes>

legal notes
=================
| SPDX-FileCopyrightText: © 2022 ekvip automation GmbH <info@ekvip.de>
| SPDX-License-Identifier: Apache-2.0
| For details check: Apache-2.0_

.. _Apache-2.0: https://www.apache.org/licenses/LICENSE-2.0

.. </legal notes>

parameters
=================

InOut:
	+-----------------+------+---------+------+------------------------------------------+
	| Scope           | Name | Type    | Init | Comment                                  |
	+=================+======+=========+======+==========================================+
	| Output CONSTANT | NULL | __XWORD | 0    | ``NULL`` is a constant which is always 0 |
	+-----------------+------+---------+------+------------------------------------------+

*)
METHOD deepDestruct
VAR_OUTPUT CONSTANT
	(* NULL is a constant which is always 0 *)
	NULL	: __XWORD := 0;
END_VAR
VAR
	indexY:UDINT;
	indexX:UDINT;
END_VAR
FOR indexY := 0 TO THIS^.dim1-1 DO
	FOR indexX := 0 TO THIS^.dim2-1 DO
		IF(THIS^.container[(indexY*THIS^.dim2)+indexX] <> 0)THEN
			THIS^.container[(indexY*THIS^.dim2)+indexX].destruct();
		END_IF
	END_FOR
END_FOR
THIS^.destruct();
END_METHOD

(*FB_Exit must be implemented explicitly. If there is an implementation, then the
method is called before the controller removes the code of the function block instance
(implicit call). The return value is not evaluated.*)
METHOD FB_Exit : BOOL
VAR_INPUT
	(* TRUE: the exit method is called in order to leave the instance which will be copied afterwards (online change).  *)
	bInCopyCode	: BOOL;
END_VAR
__DELETE(THIS^.container);
END_METHOD

(*

short summary
=================
The constructor ``FB_init`` is needed to create an unique hash code.
The hash code is a pseudo random number create with a xorshift_ algorithm.
It can be overwritten on derivations, because it will be called implicit, ``SUPER^.FB_init()`` is not required.
For more information check: `Behavoir with derived function blocks`_

.. _Behavoir with derived function blocks: https://infosys.beckhoff.com/content/1033/tc3_plc_intro/5482088715.html?id=6983869892358031022
.. _xorshift: https://en.wikipedia.org/wiki/Xorshift

.. <legal notes>

legal notes
=================
| SPDX-FileCopyrightText: © 2022 ekvip automation GmbH <info@ekvip.de>
| SPDX-License-Identifier: Apache-2.0
| For details check: Apache-2.0_

.. _Apache-2.0: https://www.apache.org/licenses/LICENSE-2.0

.. </legal notes>

parameters
=================

*)
METHOD FB_init : BOOL
VAR_INPUT
	(* if TRUE, the retain variables are initialized (warm start / cold start)*)
	bInitRetains	: BOOL;
	(* if TRUE, the instance afterwards gets moved into the copy code (online change) *)
	bInCopyCode	: BOOL;
	sizeDim1 :UDINT;
	sizeDim2 :UDINT;
END_VAR
THIS^.container := __NEW(__XWORD, (sizeDim1 * sizeDim2));
THIS^.dim1 := sizeDim1;
THIS^.dim2 := sizeDim2;
END_METHOD

METHOD getObjectAt : IObject
VAR_INPUT
	y :UDINT; //dimension 1
	x :UDINT; //dimension 2
END_VAR
getObjectAt := THIS^.container[(y*THIS^.dim2)+x];
END_METHOD

METHOD isInBounds : BOOL
VAR_INPUT
	x :UDINT;
	y :UDINT;
END_VAR
isInBounds := (x < THIS^.dim2 AND y < THIS^.dim1); //cheat >= 0 by UDINT overflow
END_METHOD

METHOD setObjectAt
VAR_INPUT
	y :UDINT; //dimension 1
	x :UDINT; //dimension 2
	obj :CNM_AbstractObject.IObject;
END_VAR
THIS^.container[(y*THIS^.dim2)+x] := obj;
END_METHOD

END_FUNCTION_BLOCK

// ---- Day05/Day05Solution.TcPOU
FUNCTION_BLOCK Day05Solution EXTENDS AbstractSolver

METHOD solve
VAR_INPUT
	step	: DINT;
END_VAR
VAR_INST
	pathInserted :BOOL;
	pageOrders :CNM_Collections.ArrayList(1000);
	pages :ARRAY[0..1000] OF IPage;
	pageList1 :CNM_Collections.ArrayList(10);
	pageList2 :CNM_Collections.ArrayList(10);
	prints :CNM_Collections.ArrayList(100);	
	currentParseList :CNM_CollectionInterfaces.IArrayList;
	parser :NumberParser();
	sum : DINT;
	sum2 : DINT;
END_VAR
VAR
	valid :BOOL;
	parsed :CNM_CollectionInterfaces.IArrayList;
	tmpObj :CNM_AbstractObject.IObject;
	tmpValue:CNM_AoC.IHaveValue;
	tmpPage :IPage;
	tmpPage2 :IPage;
	page1 :LREAL;
	page2 :LREAL;
	pPage :POINTER TO Page;
	print :CNM_CollectionInterfaces.IArrayList;
	pageOrder :CNM_CollectionInterfaces.IArrayList;
	sequenceCopy :CNM_CollectionInterfaces.IArrayList;
	index : DINT;
	currentLine :ILine;
	currentLineObject :IObject;
END_VAR
VAR CONSTANT
	READ_INPUT :DINT := 2;
	GET_LINES :DINT := READ_INPUT + 1;
	PARSE :DINT := GET_LINES + 1;
	PARSE_PAGES :DINT := PARSE + 1;
	SOLVE_PART12 :DINT := PARSE_PAGES + 1;
	APPEND_SOLUTION :DINT := SOLVE_PART12 + 1;
	WRITE_SOLUTION :DINT := APPEND_SOLUTION + 1;
	CLEAN_UP :DINT := WRITE_SOLUTION + 1;
END_VAR
CASE step OF
PARSE:	
	currentParseList := pageOrders;
	THIS^.lines.iterate(execute := FALSE);
	WHILE(THIS^.lines.iterate(execute := TRUE, line => currentLine) = CNM_ReturnTypes.SingleExecutionState.BUSY)DO
		IF(LEN(currentLine.text) = 0)THEN
			currentParseList := prints;
			CONTINUE;
		END_IF
		parsed := parser.getAllNumbers(currentLine);
		IF(parsed.size > 2 AND currentParseList.hashcode <> prints.hashcode)THEN
			currentParseList := prints;			
		END_IF
		currentParseList.append(parsed);
	END_WHILE
	cm.proceed();	
PARSE_PAGES:
	cm.evaluate(pageOrders.iterate(cm.executeStep, object => tmpObj));
	IF(__QUERYINTERFACE(tmpObj, pageOrder))THEN
		pageOrder.getObjectAt(0, object => tmpObj);
		__QUERYINTERFACE(tmpObj, tmpValue);
		page1 := (tmpValue.value);
		pageOrder.getObjectAt(1, object => tmpObj);
		__QUERYINTERFACE(tmpObj, tmpValue);
		page2 := (tmpValue.value);
		
		IF(pages[TO_DINT(page1)] <> 0)THEN
			pages[TO_DINT(page1)].addSuccessor(tmpValue);
		ELSE
			pPage := __NEW(Page(value := page1));
			__QUERYINTERFACE(pPage^, pages[TO_DINT(page1)]);
			pages[TO_DINT(page1)].addSuccessor(tmpValue);
		END_IF
	END_IF	
SOLVE_PART12:
	cm.evaluate(prints.iterate(cm.executeStep, object => tmpObj));
	IF(__QUERYINTERFACE(tmpObj, print))THEN
		pageList1.clear();
		pageList2.clear();
		print.iterate(FALSE);
		WHILE(print.iterate(TRUE, object => tmpObj) = CNM_ReturnTypes.SingleExecutionState.BUSY AND_THEN __QUERYINTERFACE(tmpObj, tmpValue))DO
			pageList1.append(pages[TO_DINT(tmpValue.value)]);
			pageList2.append(pages[TO_DINT(tmpValue.value)]);
		END_WHILE
		pageList2.instant.sort();	
		valid := TRUE;
		FOR index := 0 TO TO_DINT(pageList1.size)-1 DO
			pageList1.getObjectAt(index, object => tmpObj);
			__QUERYINTERFACE(tmpObj, tmpPage);
			pageList2.getObjectAt(index, object => tmpObj);
			__QUERYINTERFACE(tmpObj, tmpPage2);
			valid := valid AND tmpPage.isEqual(tmpPage2);
		END_FOR
		pageList2.getObjectAt((pageList2.size-1)/2, object => tmpObj);
		__QUERYINTERFACE(tmpObj, tmpPage2);
		IF(valid)THEN			
			sum := sum + TO_DINT(tmpPage2.value);
		ELSE
			sum2 := sum2 + TO_DINT(tmpPage2.value);			
		END_IF
	END_IF		
APPEND_SOLUTION:
	THIS^.bufferWrite :=Concat(THIS^.bufferWrite, Concat(TO_STRING(sum), '$n'));
	THIS^.bufferWrite :=Concat(THIS^.bufferWrite, Concat(TO_STRING(sum2), '$n'));
	cm.proceed();
WRITE_SOLUTION:
	THIS^.writeSolution();
CLEAN_UP:
	cm.step.next := CNM_ReturnTypes.DefaultSteps.STEP.SUCCESS;
	lines.deepDestruct();
	pageOrders.deepDestruct();
	cm.proceed();
END_CASE
END_METHOD

END_FUNCTION_BLOCK

// ---- Day05/Page.TcPOU
{attribute 'enable_dynamic_creation'}
FUNCTION_BLOCK Page EXTENDS Object IMPLEMENTS IPage
VAR
	myValue :LREAL;
	mySuccessors :CNM_Collections.ArrayList(50);
END_VAR

METHOD addSuccessor
VAR_INPUT
	successor	: CNM_AoC.IHaveValue;
END_VAR
THIS^.mySuccessors.append(successor);
END_METHOD

(*

short summary
=================
This abstract property returns the class name of the concrete object, 
which is useful for logging/debugging purpose or to check the class name
for ``__DELETE`` in factories (sometimes it's necessary to do more 
than just to free the memory).

.. <legal notes>

legal notes
=================
| SPDX-FileCopyrightText: © 2022 ekvip automation GmbH <info@ekvip.de>
| SPDX-License-Identifier: Apache-2.0
| For details check: Apache-2.0_

.. _Apache-2.0: https://www.apache.org/licenses/LICENSE-2.0

.. </legal notes>

*)
PROPERTY className : CNM_AbstractObject.ClassName
GET
className := 'Page';
END_GET
END_PROPERTY

(*

short summary
=================
This method compares a foreign object with the own one, this is needed for sort orders.

.. <legal notes>

legal notes
=================
| SPDX-FileCopyrightText: © 2022 ekvip automation GmbH <info@ekvip.de>
| SPDX-License-Identifier: Apache-2.0
| For details check: Apache-2.0_

.. _Apache-2.0: https://www.apache.org/licenses/LICENSE-2.0

.. </legal notes>

parameters
=================
:return:``SMALLER``: ``THIS`` precedes in order,
``EQUAL``: ``THIS`` and ``object`` at the same position in order,
``GREATER``: ``THIS`` is after in order.
Checkout the library CNM_ReturnTypes.

*)
METHOD compareTo : CNM_AbstractObject.CNM_ReturnTypes.ComparationResult
VAR_INPUT
	(* foreign objet to compare*)
	object	: CNM_AbstractObject.IObject;
END_VAR
VAR
	other :CNM_AoC.IHaveValue;
END_VAR
IF(__QUERYINTERFACE(object, other))THEN
	IF(THIS^.mySuccessors.containsEqualObject(other))THEN
		compareTo := CNM_ReturnTypes.ComparationResult.SMALLER;
	ELSIF(THIS^.value = (other.value))THEN		
		compareTo := CNM_ReturnTypes.ComparationResult.EQUAL;
	ELSE		
		compareTo := CNM_ReturnTypes.ComparationResult.GREATER;
	END_IF
ELSE
	compareTo := CNM_ReturnTypes.ComparationResult.SMALLER;
END_IF
END_METHOD

(*

short summary
=================
The constructor ``FB_init`` is needed to create an unique hash code.
The hash code is a pseudo random number create with a xorshift_ algorithm.
It can be overwritten on derivations, because it will be called implicit, ``SUPER^.FB_init()`` is not required.
For more information check: `Behavoir with derived function blocks`_

.. _Behavoir with derived function blocks: https://infosys.beckhoff.com/content/1033/tc3_plc_intro/5482088715.html?id=6983869892358031022
.. _xorshift: https://en.wikipedia.org/wiki/Xorshift

.. <legal notes>

legal notes
=================
| SPDX-FileCopyrightText: © 2022 ekvip automation GmbH <info@ekvip.de>
| SPDX-License-Identifier: Apache-2.0
| For details check: Apache-2.0_

.. _Apache-2.0: https://www.apache.org/licenses/LICENSE-2.0

.. </legal notes>

parameters
=================

*)
METHOD FB_init : BOOL
VAR_INPUT
	(* if TRUE, the retain variables are initialized (warm start / cold start)*)
	bInitRetains	: BOOL;
	(* if TRUE, the instance afterwards gets moved into the copy code (online change) *)
	bInCopyCode	: BOOL;
	value :LREAL;
END_VAR
THIS^.myValue := value;
END_METHOD

PROPERTY value : LREAL
GET
value := THIS^.myValue;
END_GET
SET
END_SET
END_PROPERTY

END_FUNCTION_BLOCK

// ---- Day06/Day06Solution.TcPOU
FUNCTION_BLOCK Day06Solution EXTENDS AbstractSolver

METHOD solve
VAR_INPUT
	step	: DINT;
END_VAR
VAR_INST
	sum : DINT;
	badGuyGuard :Guard();
	loopY :DINT;
END_VAR
VAR_INST
	guardStartX :DINT;
	guardStartY :DINT;
END_VAR
VAR_INST //map stuff	
	sizeY :UDINT;
	sizeX :UDINT;
	map :I2dArray;
	pMap :POINTER TO Dynamic2dArray;
	indexX :DINT;
	indexY :DINT;
	lineText :Tc2_System.T_MaxString;
	curChar :STRING(1);
	pVal :POINTER TO CNM_AoC.Value;
END_VAR
VAR
	parsed :CNM_CollectionInterfaces.IArrayList;
	tmpObj :CNM_AbstractObject.IObject;
	tmpVal :CNM_AoC.IHaveValue;
	sequence :CNM_CollectionInterfaces.IArrayList;
	sequenceCopy :CNM_CollectionInterfaces.IArrayList;
	index : DINT;
	currentLine :ILine;
	currentLineObject :IObject;
END_VAR
VAR CONSTANT
	READ_INPUT :DINT := 2;
	GET_LINES :DINT := READ_INPUT + 1;
	PARSE :DINT := GET_LINES + 1;
	SOLVE_PART1 :DINT := PARSE + 1;
	RESET_FOR_PART2 :DINT := SOLVE_PART1 + 1;
	SOLVE_PART2 :DINT := RESET_FOR_PART2 + 1;
	APPEND_SOLUTION :DINT := SOLVE_PART2 + 1;
	WRITE_SOLUTION :DINT := APPEND_SOLUTION + 1;
	CLEAN_UP :DINT := WRITE_SOLUTION + 1;
END_VAR
CASE step OF
PARSE:	
	lines.getLineAt(0, line => currentLine);
	sizeY := TO_UDINT(lines.size);
	sizeX := LEN(currentLine.text);
	pMap := __NEW(Dynamic2dArray(sizeDim1 := sizeY, sizeDim2 := sizeX));
	RETURN (NOT __QUERYINTERFACE(pMap^,map));
	THIS^.lines.iterate(execute := FALSE);
	indexY := 0;
	WHILE(THIS^.lines.iterate(execute := TRUE, line => currentLine) = CNM_ReturnTypes.SingleExecutionState.BUSY)DO
		FOR index := 0 TO sizeX-1 DO
			lineText := currentLine.text;
			curChar := F_ToCHR(lineText[index]);
			IF(curChar = '.')THEN				
				pVal := __NEW(Value());
				pVal^.value := 0;
				map.setObjectAt(y := indexY, x := index, pVal^);
			ELSIF(curChar = '#')THEN				
				pVal := __NEW(Value());
				pVal^.value := 1;
				map.setObjectAt(y := indexY, x := index, pVal^);
			ELSIF(curChar = '^')THEN				
				pVal := __NEW(Value());
				pVal^.value := 0;
				badGuyGuard.x := index;
				badGuyGuard.y := indexY;
				badGuyGuard.direction := Rotation.UP;
				guardStartX := index;
				guardStartY := indexY;
				map.setObjectAt(y := indexY, x := index, pVal^);
			END_IF
		END_FOR
		indexY := indexY+1;
	END_WHILE
	cm.proceed();
SOLVE_PART1:
	THIS^.walkToEdge(guard := badGuyGuard, map := map, maxX := sizeX, maxY := sizeY, visitedFields => sum);
	cm.proceed();	
RESET_FOR_PART2:
	THIS^.bufferWrite := Concat(TO_STRING(sum), '$n');
	sum := 0;
	cm.proceed();
	indexY := 0;
SOLVE_PART2:
	FOR index := 0 TO sizeX-1 DO
		IF(index = guardStartX AND indexY = guardStartY)THEN
			CONTINUE;
		END_IF
		tmpObj := map.getObjectAt(x := index, y := indexY);
		IF(__QUERYINTERFACE(tmpObj, tmpVal) AND_THEN tmpVal.value = 0)THEN		
			tmpVal.value := 1; //set stone
			badGuyGuard.x := guardStartX;
			badGuyGuard.y := guardStartY;
			badGuyGuard.direction := Rotation.UP;
			sum := sum + SEL(THIS^.walkToEdge(guard := badGuyGuard, map := map, maxX := sizeX, maxY := sizeY, visitedFields => sum), 1, 0);
			tmpVal.value := 0; //reset stone
		END_IF
	END_FOR	
	indexY := indexY+1;
	cm.waitFor(indexY = sizeY);
APPEND_SOLUTION:
	THIS^.bufferWrite :=Concat(THIS^.bufferWrite, Concat(TO_STRING(sum), '$n'));
	cm.proceed();
WRITE_SOLUTION:
	THIS^.writeSolution();
CLEAN_UP:
	cm.step.next := CNM_ReturnTypes.DefaultSteps.STEP.SUCCESS;
	lines.deepDestruct();
	map.deepDestruct();
	cm.proceed();
END_CASE
END_METHOD

METHOD walkToEdge : BOOL //false if loop
VAR_INPUT
	guard :IGuard;
	map :I2dArray;
	maxX :DINT;
	maxY :DINT;
END_VAR
VAR_OUTPUT
	visitedFields :DINT;
END_VAR
VAR
	seenField :BOOL;
	index :DINT;
	//there is no dictionary yet so I am just lazy and will do this:
	//could also just be a list with contains, but naaahhh
	seen :ARRAY[0..255,0..255,0..3] OF BOOL; //x, y, rotation
END_VAR
WHILE(guard.x <> 0 AND_THEN guard.x <> maxX-1 AND_THEN guard.y <> 0 AND_THEN guard.y <> maxY-1)DO
	RETURN (seen[guard.x, guard.y, guard.direction]);
	seenField := FALSE;
	FOR index := 0 TO 3 DO
		IF(seen[guard.x, guard.y, index])THEN
			seenField := TRUE;
		END_IF
	END_FOR
	visitedFields := visitedFields + SEL(seenField, 1, 0); //only add fields which where never seen
	seen[guard.x, guard.y, guard.direction] := TRUE;
	guard.walk(map);
END_WHILE

visitedFields := visitedFields + 1; //add the last field, or replace with repeat loop
walkToEdge := TRUE;
END_METHOD

END_FUNCTION_BLOCK

// ---- Day06/Guard/Guard.TcPOU
FUNCTION_BLOCK Guard EXTENDS Object IMPLEMENTS IGuard
VAR
	myX :DINT;
	myY :DINT;
	myRotation :Rotation;
	up :MoveUp();
	right :MoveRight();
	down :MoveDown();
	left :MoveLeft();
	myMoves :ARRAY[0..3] OF IMove := [up, right, down, left];
END_VAR

(*

short summary
=================
This abstract property returns the class name of the concrete object, 
which is useful for logging/debugging purpose or to check the class name
for ``__DELETE`` in factories (sometimes it's necessary to do more 
than just to free the memory).

.. <legal notes>

legal notes
=================
| SPDX-FileCopyrightText: © 2022 ekvip automation GmbH <info@ekvip.de>
| SPDX-License-Identifier: Apache-2.0
| For details check: Apache-2.0_

.. _Apache-2.0: https://www.apache.org/licenses/LICENSE-2.0

.. </legal notes>

*)
PROPERTY className : CNM_AbstractObject.ClassName
GET
className := 'Guard';
END_GET
END_PROPERTY

PROPERTY direction : Rotation
GET
direction := THIS^.myRotation;
END_GET
SET
THIS^.myRotation := direction;
END_SET
END_PROPERTY

METHOD walk
VAR_INPUT
	map	: I2dArray;
END_VAR
VAR
	currentDirection :DINT;
END_VAR
currentDirection := THIS^.direction;

WHILE(NOT THIS^.myMoves[currentDirection].tryMove(THIS^, map))DO
	currentDirection := (currentDirection + 1) MOD 4; //rotate right
END_WHILE
END_METHOD

PROPERTY x : DINT
GET
x := THIS^.myX;
END_GET
SET
THIS^.myX := x;
END_SET
END_PROPERTY

PROPERTY y : DINT
GET
y := THIS^.myY;
END_GET
SET
THIS^.myY := y;
END_SET
END_PROPERTY

END_FUNCTION_BLOCK

// ---- Day06/Moves/MoveUp.TcPOU
FUNCTION_BLOCK MoveUp EXTENDS GuardMove
VAR_INPUT
END_VAR
VAR_OUTPUT
END_VAR
VAR
END_VAR

(*

short summary
=================
This abstract property returns the class name of the concrete object, 
which is useful for logging/debugging purpose or to check the class name
for ``__DELETE`` in factories (sometimes it's necessary to do more 
than just to free the memory).

.. <legal notes>

legal notes
=================
| SPDX-FileCopyrightText: © 2022 ekvip automation GmbH <info@ekvip.de>
| SPDX-License-Identifier: Apache-2.0
| For details check: Apache-2.0_

.. _Apache-2.0: https://www.apache.org/licenses/LICENSE-2.0

.. </legal notes>

*)
PROPERTY className : CNM_AbstractObject.ClassName
GET
className := 'MoveUp';
END_GET
END_PROPERTY

PROPERTY PROTECTED direction : Rotation
GET
direction := Rotation.UP;
END_GET
END_PROPERTY

END_FUNCTION_BLOCK

// ---- Day06/Moves/GuardMove.TcPOU
FUNCTION_BLOCK ABSTRACT GuardMove EXTENDS Object IMPLEMENTS IMove

(*

short summary
=================
This abstract property returns the class name of the concrete object, 
which is useful for logging/debugging purpose or to check the class name
for ``__DELETE`` in factories (sometimes it's necessary to do more 
than just to free the memory).

.. <legal notes>

legal notes
=================
| SPDX-FileCopyrightText: © 2022 ekvip automation GmbH <info@ekvip.de>
| SPDX-License-Identifier: Apache-2.0
| For details check: Apache-2.0_

.. _Apache-2.0: https://www.apache.org/licenses/LICENSE-2.0

.. </legal notes>

*)
PROPERTY className : CNM_AbstractObject.ClassName
GET
END_GET
END_PROPERTY

PROPERTY PROTECTED ABSTRACT direction : Rotation
GET
END_GET
END_PROPERTY

METHOD getMoveOffset : BOOL
VAR_OUTPUT
	x :DINT;
	y:DINT;
END_VAR
CASE THIS^.direction OF
Rotation.UP:
	x := 0;
	y := -1;
Rotation.RIGHT:
	x := 1;
	y := 0;
Rotation.DOWN:
	x := 0;
	y := 1;
Rotation.LEFT:
	x := -1;
	y := 0;
END_CASE
END_METHOD

METHOD tryMove : BOOL
VAR_INPUT
	guard :IGuard;
	map	: I2dArray;
	collision :DINT := 1;
END_VAR
VAR
	diffX :DINT;
	diffY :DINT;
	newX :DINT;
	newY :DINT;
	obj :CNM_AbstractObject.IObject;
	val :CNM_AoC.IHaveValue;
END_VAR
THIS^.getMoveOffset(x => diffX, y => diffY);
newX := guard.x + diffX;
newY := guard.y + diffY;

tryMove := FALSE;

RETURN(NOT map.isInBounds(x := newX, y := newY));

obj := map.getObjectAt(x := newX, y := newY);

IF(__QUERYINTERFACE(obj, val) AND_THEN TO_DINT(val.value) <> collision)THEN
	tryMove := TRUE;
	guard.x := newX;
	guard.y := newY;
	guard.direction := THIS^.direction;
END_IF
END_METHOD

END_FUNCTION_BLOCK

// ---- Day06/Moves/MoveRight.TcPOU
FUNCTION_BLOCK MoveRight EXTENDS GuardMove
VAR_INPUT
END_VAR
VAR_OUTPUT
END_VAR
VAR
END_VAR

(*

short summary
=================
This abstract property returns the class name of the concrete object, 
which is useful for logging/debugging purpose or to check the class name
for ``__DELETE`` in factories (sometimes it's necessary to do more 
than just to free the memory).

.. <legal notes>

legal notes
=================
| SPDX-FileCopyrightText: © 2022 ekvip automation GmbH <info@ekvip.de>
| SPDX-License-Identifier: Apache-2.0
| For details check: Apache-2.0_

.. _Apache-2.0: https://www.apache.org/licenses/LICENSE-2.0

.. </legal notes>

*)
PROPERTY className : CNM_AbstractObject.ClassName
GET
className := 'MoveRight';
END_GET
END_PROPERTY

PROPERTY PROTECTED direction : Rotation
GET
direction := Rotation.RIGHT;
END_GET
END_PROPERTY

END_FUNCTION_BLOCK

// ---- Day06/Moves/MoveDown.TcPOU
FUNCTION_BLOCK MoveDown EXTENDS GuardMove
VAR_INPUT
END_VAR
VAR_OUTPUT
END_VAR
VAR
END_VAR

(*

short summary
=================
This abstract property returns the class name of the concrete object, 
which is useful for logging/debugging purpose or to check the class name
for ``__DELETE`` in factories (sometimes it's necessary to do more 
than just to free the memory).

.. <legal notes>

legal notes
=================
| SPDX-FileCopyrightText: © 2022 ekvip automation GmbH <info@ekvip.de>
| SPDX-License-Identifier: Apache-2.0
| For details check: Apache-2.0_

.. _Apache-2.0: https://www.apache.org/licenses/LICENSE-2.0

.. </legal notes>

*)
PROPERTY className : CNM_AbstractObject.ClassName
GET
className := 'MoveDown';
END_GET
END_PROPERTY

PROPERTY PROTECTED direction : Rotation
GET
direction := Rotation.DOWN;
END_GET
END_PROPERTY

END_FUNCTION_BLOCK

// ---- Day06/Moves/MoveLeft.TcPOU
FUNCTION_BLOCK MoveLeft EXTENDS GuardMove
VAR_INPUT
END_VAR
VAR_OUTPUT
END_VAR
VAR
END_VAR

(*

short summary
=================
This abstract property returns the class name of the concrete object, 
which is useful for logging/debugging purpose or to check the class name
for ``__DELETE`` in factories (sometimes it's necessary to do more 
than just to free the memory).

.. <legal notes>

legal notes
=================
| SPDX-FileCopyrightText: © 2022 ekvip automation GmbH <info@ekvip.de>
| SPDX-License-Identifier: Apache-2.0
| For details check: Apache-2.0_

.. _Apache-2.0: https://www.apache.org/licenses/LICENSE-2.0

.. </legal notes>

*)
PROPERTY className : CNM_AbstractObject.ClassName
GET
className := 'MoveLeft';
END_GET
END_PROPERTY

PROPERTY PROTECTED direction : Rotation
GET
direction := Rotation.LEFT;
END_GET
END_PROPERTY

END_FUNCTION_BLOCK

// ---- Day07/Day07Solution.TcPOU
FUNCTION_BLOCK Day07Solution EXTENDS AbstractSolver

METHOD concatVals : ULINT
VAR_INPUT
	left :ULINT;
	right :ULINT;
END_VAR
VAR
	log10 :LREAL;
END_VAR
log10 := LOG(right);

concatVals := left * TO_ULINT(EXPT(10, THIS^.roundUp(log10))) + right;

IF(concatVals < left * right)THEN
	concatVals := 0; //error
END_IF
END_METHOD

METHOD roundUp : ULINT
VAR_INPUT
	value :LREAL;
END_VAR
VAR
	up :ULINT;
END_VAR
roundUp := TRUNC(value)+1;
END_METHOD

METHOD solve
VAR_INPUT
	step	: DINT;
END_VAR
VAR_INST
	pathInserted :BOOL;
	sequences :CNM_Collections.ArrayList(100);
	parser :NumberParser();
	sum : ULINT;
	goal :ULINT;
END_VAR
VAR
	parsed :CNM_CollectionInterfaces.IArrayList;
	tmpObj :CNM_AbstractObject.IObject;
	tmpVal :CNM_AoC.IHaveUlintValue;
	sequence :CNM_CollectionInterfaces.IArrayList;
	sequenceCopy :CNM_CollectionInterfaces.IArrayList;
	index : DINT;
	currentLine :ILine;
	currentLineObject :IObject;
END_VAR
VAR CONSTANT
	READ_INPUT :DINT := 2;
	GET_LINES :DINT := READ_INPUT + 1;
	PARSE :DINT := GET_LINES + 1;
	SOLVE_PART1 :DINT := PARSE + 1;
	RESET_FOR_PART2 :DINT := SOLVE_PART1 + 1;
	SOLVE_PART2 :DINT := RESET_FOR_PART2 + 1;
	APPEND_SOLUTION :DINT := SOLVE_PART2 + 1;
	WRITE_SOLUTION :DINT := APPEND_SOLUTION + 1;
	CLEAN_UP :DINT := WRITE_SOLUTION + 1;
END_VAR
CASE step OF
PARSE:	
	THIS^.lines.iterate(execute := FALSE);
	WHILE(THIS^.lines.iterate(execute := TRUE, line => currentLine) = CNM_ReturnTypes.SingleExecutionState.BUSY)DO
		parsed := parser.getAllNumbersUlint(currentLine);
		sequences.append(parsed);
	END_WHILE
	cm.proceed();	
SOLVE_PART1:
	cm.evaluate(sequences.iterate(cm.executeStep, object => tmpObj));
	IF(__QUERYINTERFACE(tmpObj, sequence))THEN
		sequence.getObjectAt(0, object => tmpObj);
		IF(__QUERYINTERFACE(tmpObj, tmpVal))THEN
			goal := tmpVal.value;
			sum := sum + SEL(THIS^.trySolve(0, 1, sequence, -1, goal), 0, goal);
		END_IF
	END_IF		
RESET_FOR_PART2:
	THIS^.bufferWrite := Concat(TO_STRING(sum), '$n');
	sum := 0;
	cm.proceed();
SOLVE_PART2:
	cm.evaluate(sequences.iterate(cm.executeStep, object => tmpObj));
	IF(__QUERYINTERFACE(tmpObj, sequence))THEN
		sequence.getObjectAt(0, object => tmpObj);
		IF(__QUERYINTERFACE(tmpObj, tmpVal))THEN
			goal := tmpVal.value;
			sum := sum + SEL(THIS^.trySolve(0, 1, sequence, -1, goal, TRUE), 0, goal);
		END_IF
	END_IF		
APPEND_SOLUTION:
	THIS^.bufferWrite :=Concat(THIS^.bufferWrite, Concat(TO_STRING(sum), '$n'));
	cm.proceed();
WRITE_SOLUTION:
	THIS^.writeSolution();
CLEAN_UP:
	cm.step.next := CNM_ReturnTypes.DefaultSteps.STEP.SUCCESS;
	lines.deepDestruct();
	sequences.deepDestruct();
	cm.proceed();
END_CASE
END_METHOD

METHOD trySolve : BOOL
VAR_INPUT
	prevValue :ULINT := 0;
	index :DINT := 0;
	numbers :CNM_CollectionInterfaces.IArrayList;
	operator :DINT;
	goal :ULINT;
	part2 :BOOL := FALSE;
END_VAR
VAR
	obj :CNM_AbstractObject.IObject;
	val :CNM_AoC.IHaveUlintValue;
	curVal :ULINT;
END_VAR
IF(index >= numbers.size)THEN
	trySolve := goal = prevValue;
	RETURN;
END_IF

IF(prevValue > goal)THEN
	trySolve := FALSE;
	RETURN;
END_IF

numbers.getObjectAt(index, object => obj);
RETURN (NOT __QUERYINTERFACE(obj, val));
curVal := val.value;

IF(index = 1)THEN	
	trySolve := 
		THIS^.trySolve(curVal, index + 1, numbers, 0, goal, part2)
		OR THIS^.trySolve(curVal, index + 1, numbers, 1, goal, part2)
		OR part2 AND_THEN THIS^.trySolve(curVal, index + 1, numbers, 2, goal, part2);
	RETURN;
END_IF

CASE operator OF
0: //+
	trySolve := 
		THIS^.trySolve(prevValue+curVal, index + 1, numbers, 0, goal, part2)
		OR THIS^.trySolve(prevValue+curVal, index + 1, numbers, 1, goal, part2)
		OR part2 AND_THEN THIS^.trySolve(prevValue+curVal, index + 1, numbers, 2, goal, part2);
1: //*
	trySolve := 
		THIS^.trySolve(prevValue*curVal, index + 1, numbers, 0, goal, part2)
		OR THIS^.trySolve(prevValue*curVal, index + 1, numbers, 1, goal, part2)
		OR part2 AND_THEN THIS^.trySolve(prevValue*curVal, index + 1, numbers, 2, goal, part2);
2: // ||
	trySolve := 
		THIS^.trySolve(THIS^.concatVals(prevValue,curVal), index + 1, numbers, 0, goal, part2)
		OR THIS^.trySolve(THIS^.concatVals(prevValue,curVal), index + 1, numbers, 1, goal, part2)
		OR part2 AND_THEN THIS^.trySolve(THIS^.concatVals(prevValue,curVal), index + 1, numbers, 2, goal, part2);
END_CASE
END_METHOD

END_FUNCTION_BLOCK
